// TIA Portal V19 export
TYPE "C501_VAR_IF_TRA_TYPIC"
   STRUCT
      EXT_HW { ExternalAccessible := 'False'; ExternalVisible := 'False'; ExternalWritable := 'False'} : Bool;   // Sturings hardware (PLC) in storing
      STO { ExternalAccessible := 'False'; ExternalVisible := 'False'; ExternalWritable := 'False'} : Struct   // Opsomming van alle storingen
         A001 : Bool;   // Storing vorstbeveiliging
      END_STRUCT;
   END_STRUCT;
END_TYPE
